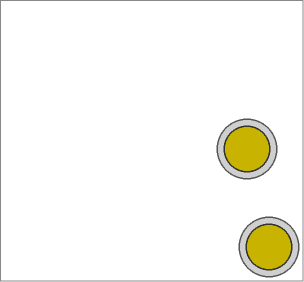
VISUALIZATION Visualization  // 304x282
    Lamp1 (212,114 70x70), variable: Main.KlaarVoorBier, style: Lamp-Lamp1-Yellow
    Lamp1 (234,212 70x70), variable: Main.KlaarVoorSpel, style: Lamp-Lamp1-Yellow
END_VISUALIZATION

(* stored: Version 1.1.0.1, ProductVersion 3.1.4024.15
   Visu Visualization: Id {20cfc91b-0b5a-4222-add0-263ef55ba61c} *)
